FUNCTION FC_HeatingCurve : REAL
VAR_INPUT
	fTempAmb 	: REAL; 		//Ambient temperature
	fSlope 		: REAL := -1; 	//Slope of heatcurve
	fOffset 	: REAL := 36;	//In °C; off set at T_amb=0°C
END_VAR
VAR
END_VAR
VAR CONSTANT 
END_VAR

FC_HeatingCurve := fSlope * fTempAmb + fOffset;

END_FUNCTION

(* stored: Version 1.1.0.1, ProductVersion 3.1.4024.6
   POU FC_HeatingCurve: Id {dc111241-9f5f-4341-81b4-6d748baebe02}, SpecialFunc None *)
